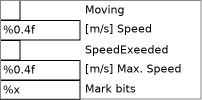
VISUALIZATION _VISU_MachineOut  // 202x100
VAR_IN_OUT
	ref : ST_ModuleMachineInterface_OUT;
END_VAR
    Rectangle (0,20 80x20), "%0.4f", text variable: ref.fSpeed
    Rectangle (82,20 120x18), "[m/s] Speed"
    Rectangle (0,60 80x20), "%0.4f", text variable: ref.fMaxSpeed
    Rectangle (82,60 120x18), "[m/s] Max. Speed"
    Rectangle (82,0 120x20), "Moving"
    RoundedRectangle (0,40 20x20), colour toggle: ref.bSpeedExeeded
    Rectangle (82,40 120x20), "SpeedExeeded"
    RoundedRectangle (0,0 20x20), colour toggle: ref.bMoving
    Rectangle (0,80 80x20), "%x", text variable: ref.nPrintMarkPosBits
    Rectangle (82,80 120x18), "Mark bits"
END_VISUALIZATION

(* stored: Version 1.1.0.1, ProductVersion 3.1.4024.11
   Visu _VISU_MachineOut: Id {c8a08db4-c54a-4e88-820a-73a613c7186c} *)
